TYPE TRACK:
STRUCT
	//Mainly for WInch control and boxcar sim

	red_left: REAL := 0.426085;
	red_right: REAL:= 35.377296;
	red_middle: REAL:= 17.887;
	blue_left: REAL:= 7.244;
	blue_right: REAL:= 42.17;
	blue_middle: REAL:=24.681;
	sel_val: SINT := 0;
	target: REAL;
	redSelect: BOOL;
	blueSelect:BOOL;
	leftSelect:BOOL;
	rightSelect: BOOL;
	redFWD: BOOL;
	redREV: BOOL;
	blueFWD: BOOL;
	blueREV: BOOL;
	redPx: REAL;
	redPy: REAL;
	bluePx: REAL; //move with car in ignition
	bluePy: REAL; // winch position extend retract
	redREVok: BOOL;
	blueREVok: BOOL; // ok to move car onto sled
	redAttached: BOOL;
	blueAttached: BOOL;
	maxPy: REAL := 338; //max extend of winch
	minPY: REAL := 21;
	blueExtended : BOOL;
	redExtended : BOOL;
	cmdAttachRed: BOOL;
	cmdDetachRed: BOOL;
	cmdAttachBlue: BOOL;
	cmdDetachBlue: BOOL;
	
END_STRUCT
END_TYPE

(* stored: Version 1.1.0.1
   DUT TRACK: Id {d8787df0-78f8-4b2a-8c78-8e0d3c65219c} *)
